LIN {X 0,Y 68.239,Z 470.992,A -85,B 0,C 180,E1 -29740.841,E2 -29740.841} C_VEL
LIN {X 0,Y 69.162,Z 475.21,A -85,B 0,C 180,E1 -29748.344,E2 -29748.344} C_VEL
LIN {X 0,Y 69.85,Z 480.054,A -85,B 0,C 180,E1 -29755.151,E2 -29755.151} C_VEL
LIN {X 0,Y 70.329,Z 485.314,A -85,B 0,C 180,E1 -29761.664,E2 -29761.664} C_VEL
LIN {X 0,Y 70.246,Z 486.749,A -85,B 0,C 180,E1 -29763.244,E2 -29763.244} C_VEL
LIN {X 0,Y 62.959,Z 496.336,A -85,B 0,C 180,E1 -29768.731,E2 -29768.731} C_VEL
LIN {X 0,Y 56.259,Z 504.164,A -85,B 0,C 180,E1 -29775.534,E2 -29775.534} C_VEL
LIN {X 0,Y 50.423,Z 510.748,A -85,B 0,C 180,E1 -29784.262,E2 -29784.262} C_VEL
LIN {X 0,Y 45.973,Z 515.938,A -85,B 0,C 180,E1 -29794.386,E2 -29794.386} C_VEL
LIN {X 0,Y 42.364,Z 521.062,A -85,B 0,C 180,E1 -29809.38,E2 -29809.38} C_VEL
LIN {X 0,Y 41.451,Z 524.116,A -85,B 0,C 180,E1 -29822.031,E2 -29822.031} C_VEL
LIN {X 0,Y 43.45,Z 527.149,A -85,B 0,C 180,E1 -29839.683,E2 -29839.683} C_VEL
LIN {X 0,Y 48.615,Z 528.811,A -85,B 0,C 180,E1 -29854.297,E2 -29854.297} C_VEL
LIN {X 0,Y 55.931,Z 529.259,A -85,B 0,C 180,E1 -29865.444,E2 -29865.444} C_VEL
LIN {X 0,Y 64.604,Z 528.582,A -85,B 0,C 180,E1 -29873.754,E2 -29873.754} C_VEL
LIN {X 0,Y 74.136,Z 526.812,A -85,B 0,C 180,E1 -29879.999,E2 -29879.999} C_VEL
LIN {X 0,Y 84.097,Z 523.976,A -85,B 0,C 180,E1 -29884.595,E2 -29884.595} C_VEL
LIN {X 0,Y 85.983,Z 523.37,A -85,B 0,C 180,E1 -29885.95,E2 -29885.95} C_VEL
LIN {X 0,Y 87.239,Z 522.957,A -85,B 0,C 180,E1 -29888.38,E2 -29888.38} C_VEL
LIN {X 0,Y 87.487,Z 522.949,A -85,B 0,C 180,E1 -29891.862,E2 -29891.862} C_VEL
LIN {X 0,Y 87.094,Z 523.267,A -85,B 0,C 180,E1 -29894.695,E2 -29894.695} C_VEL
LIN {X 0,Y 86.771,Z 523.554,A -85,B 0,C 180,E1 -29896.465,E2 -29896.465} C_VEL
LIN {X 0,Y 84.907,Z 524.361,A -85,B 0,C 180,E1 -29897.846,E2 -29897.846} C_VEL
LIN {X 0,Y 75.254,Z 527.595,A -85,B 0,C 180,E1 -29900.948,E2 -29900.948} C_VEL
LIN {X 0,Y 63.005,Z 530.583,A -85,B 0,C 180,E1 -29906.826,E2 -29906.826} C_VEL
LIN {X 0,Y 51.75,Z 532.139,A -85,B 0,C 180,E1 -29915.426,E2 -29915.426} C_VEL
LIN {X 0,Y 42.308,Z 532.255,A -85,B 0,C 180,E1 -29928.357,E2 -29928.357} C_VEL
LIN {X 0,Y 36.34,Z 531.011,A -85,B 0,C 180,E1 -29947.243,E2 -29947.243} C_VEL
LIN {X 0,Y 35.092,Z 529.839,A -85,B 0,C 180,E1 -29958.444,E2 -29958.444} C_VEL
LIN {X 0,Y 35.123,Z 528.239,A -85,B 0,C 180,E1 -29969.997,E2 -29969.997} C_VEL
LIN {X 0,Y 35.704,Z 524.788,A -85,B 0,C 180,E1 -29987.17,E2 -29987.17} C_VEL
LIN {X 0,Y 38.996,Z 520.194,A -85,B 0,C 180,E1 -30002.726,E2 -30002.726} C_VEL
LIN {X 0,Y 45.724,Z 513.255,A -85,B 0,C 180,E1 -30016.89,E2 -30016.89} C_VEL
LIN {X 0,Y 53.05,Z 505.696,A -85,B 0,C 180,E1 -30025.889,E2 -30025.889} C_VEL
LIN {X 0,Y 56.999,Z 501.154,A -85,B 0,C 180,E1 -30029.662,E2 -30029.662} C_VEL
LIN {X 0,Y 61.398,Z 493.41,A -85,B 0,C 180,E1 -30036.302,E2 -30036.302} C_VEL
LIN {X 0,Y 63.78,Z 488.74,A -85,B 0,C 180,E1 -30039.696,E2 -30039.696} C_VEL
LIN {X 0,Y 64.398,Z 483.456,A -85,B 0,C 180,E1 -30045.786,E2 -30045.786} C_VEL
LIN {X 0,Y 64.825,Z 478.418,A -85,B 0,C 180,E1 -30052.055,E2 -30052.055} C_VEL
LIN {X 0,Y 64.92,Z 477.146,A -85,B 0,C 180,E1 -30053.786,E2 -30053.786} C_VEL
LIN {X 0,Y 64.579,Z 474.051,A -85,B 0,C 180,E1 -30060.001,E2 -30060.001} C_VEL
LIN {X 0,Y 63.893,Z 471.746,A -85,B 0,C 180,E1 -30068.141,E2 -30068.141} C_VEL
LIN {X 0,Y 63.705,Z 471.009,A -85,B 0,C 180,E1 -30072.747,E2 -30072.747} C_VEL
LIN {X 0,Y 63.211,Z 471.361,A -85,B 0,C 180,E1 -30079.485,E2 -30079.485} C_VEL
LIN {X 0,Y 63.047,Z 472.618,A -85,B 0,C 180,E1 -30086.907,E2 -30086.907} C_VEL
LIN {X 0,Y 63.522,Z 474.951,A -85,B 0,C 180,E1 -30095.851,E2 -30095.851} C_VEL
LIN {X 0,Y 63.895,Z 477.2,A -85,B 0,C 180,E1 -30101.298,E2 -30101.298} C_VEL
LIN {X 0,Y 64.259,Z 480.2,A -85,B 0,C 180,E1 -30107.059,E2 -30107.059} C_VEL
LIN {X 0,Y 64.466,Z 484.389,A -85,B 0,C 180,E1 -30113.662,E2 -30113.662} C_VEL
LIN {X 0,Y 64.505,Z 488.05,A -85,B 0,C 180,E1 -30118.836,E2 -30118.836} C_VEL
LIN {X 0,Y 63.381,Z 489.883,A -85,B 0,C 180,E1 -30120.07,E2 -30120.07} C_VEL
LIN {X 0,Y 55.729,Z 498.916,A -85,B 0,C 180,E1 -30125.807,E2 -30125.807} C_VEL
LIN {X 0,Y 48.757,Z 506.356,A -85,B 0,C 180,E1 -30133.247,E2 -30133.247} C_VEL
LIN {X 0,Y 42.447,Z 512.783,A -85,B 0,C 180,E1 -30143.439,E2 -30143.439} C_VEL
LIN {X 0,Y 38.014,Z 517.582,A -85,B 0,C 180,E1 -30155.306,E2 -30155.306} C_VEL
LIN {X 0,Y 34.671,Z 522.492,A -85,B 0,C 180,E1 -30173.919,E2 -30173.919} C_VEL
LIN {X 0,Y 34.527,Z 525.01,A -85,B 0,C 180,E1 -30187.639,E2 -30187.639} C_VEL
LIN {X 0,Y 37.457,Z 527.626,A -85,B 0,C 180,E1 -30205.743,E2 -30205.743} C_VEL
LIN {X 0,Y 44.328,Z 529.337,A -85,B 0,C 180,E1 -30222.045,E2 -30222.045} C_VEL
LIN {X 0,Y 52.33,Z 529.729,A -85,B 0,C 180,E1 -30232.281,E2 -30232.281} C_VEL
LIN {X 0,Y 63.259,Z 528.907,A -85,B 0,C 180,E1 -30240.821,E2 -30240.821} C_VEL
LIN {X 0,Y 72.278,Z 527.298,A -85,B 0,C 180,E1 -30245.579,E2 -30245.579} C_VEL
LIN {X 0,Y 83.302,Z 524.325,A -85,B 0,C 180,E1 -30249.714,E2 -30249.714} C_VEL
LIN {X 0,Y 85.768,Z 523.476,A -85,B 0,C 180,E1 -30250.483,E2 -30250.483} C_VEL
LIN {X 0,Y 87.552,Z 522.917,A -85,B 0,C 180,E1 -30252.094,E2 -30252.094} C_VEL
LIN {X 0,Y 87.094,Z 523.267,A -85,B 0,C 180,E1 -30254.695,E2 -30254.695} C_VEL
LIN {X 0,Y 86.085,Z 523.782,A -85,B 0,C 180,E1 -30256.223,E2 -30256.223} C_VEL
LIN {X 0,Y 83.521,Z 524.843,A -85,B 0,C 180,E1 -30257.731,E2 -30257.731} C_VEL
LIN {X 0,Y 79.236,Z 526.3,A -85,B 0,C 180,E1 -30258.909,E2 -30258.909} C_VEL
LIN {X 0,Y 75.495,Z 527.361,A -85,B 0,C 180,E1 -30259.378,E2 -30259.378} C_VEL
LIN {X 0,Y 64.083,Z 529.81,A -85,B 0,C 180,E1 -30260.093,E2 -30260.093} C_VEL
LIN {X 0,Y 58.606,Z 530.639,A -85,B 0,C 180,E1 -30261.55,E2 -30261.55} C_VEL
LIN {X 0,Y 57.584,Z 530.755,A -85,B 0,C 180,E1 -30262.052,E2 -30262.052} C_VEL
LIN {X 0,Y 47.968,Z 531.742,A -85,B 0,C 180,E1 -30268.465,E2 -30268.465} C_VEL
LIN {X 0,Y 37.285,Z 531.697,A -85,B 0,C 180,E1 -30281.061,E2 -30281.061} C_VEL
LIN {X 0,Y 29.932,Z 530.261,A -85,B 0,C 180,E1 -30301.989,E2 -30301.989} C_VEL
LIN {X 0,Y 28.199,Z 528.973,A -85,B 0,C 180,E1 -30315.565,E2 -30315.565} C_VEL
LIN {X 0,Y 28.043,Z 527.294,A -85,B 0,C 180,E1 -30329.996,E2 -30329.996} C_VEL
LIN {X 0,Y 28.995,Z 523.679,A -85,B 0,C 180,E1 -30351.316,E2 -30351.316} C_VEL
LIN {X 0,Y 33.235,Z 518.91,A -85,B 0,C 180,E1 -30369.37,E2 -30369.37} C_VEL
LIN {X 0,Y 39.922,Z 512.879,A -85,B 0,C 180,E1 -30382.385,E2 -30382.385} C_VEL
LIN {X 0,Y 47.972,Z 505.34,A -85,B 0,C 180,E1 -30391.516,E2 -30391.516} C_VEL
LIN {X 0,Y 50.877,Z 502.415,A -85,B 0,C 180,E1 -30393.874,E2 -30393.874} C_VEL
LIN {X 0,Y 53.428,Z 498.975,A -85,B 0,C 180,E1 -30397.035,E2 -30397.035} C_VEL
LIN {X 0,Y 57.849,Z 491.973,A -85,B 0,C 180,E1 -30402.88,E2 -30402.88} C_VEL
LIN {X 0,Y 58.451,Z 490.648,A -85,B 0,C 180,E1 -30404.124,E2 -30404.124} C_VEL
LIN {X 0,Y 59.603,Z 485.201,A -85,B 0,C 180,E1 -30411.247,E2 -30411.247} C_VEL
LIN {X 0,Y 60.222,Z 481.579,A -85,B 0,C 180,E1 -30416.656,E2 -30416.656} C_VEL
LIN {X 0,Y 60.25,Z 480.054,A -85,B 0,C 180,E1 -30420.001,E2 -30420.001} C_VEL
LIN {X 0,Y 59.924,Z 478.006,A -85,B 0,C 180,E1 -30426.736,E2 -30426.736} C_VEL
LIN {X 0,Y 59.645,Z 477,A -85,B 0,C 180,E1 -30433.631,E2 -30433.631} C_VEL
LIN {X 0,Y 59.095,Z 477.547,A -85,B 0,C 180,E1 -30440.904,E2 -30440.904} C_VEL
LIN {X 0,Y 58.901,Z 478.853,A -85,B 0,C 180,E1 -30448.508,E2 -30448.508} C_VEL
LIN {X 0,Y 59.072,Z 480.036,A -85,B 0,C 180,E1 -30453.616,E2 -30453.616} C_VEL
LIN {X 0,Y 59.17,Z 482.171,A -85,B 0,C 180,E1 -30459.622,E2 -30459.622} C_VEL
LIN {X 0,Y 59.182,Z 485.792,A -85,B 0,C 180,E1 -30467.178,E2 -30467.178} C_VEL
LIN {X 0,Y 58.934,Z 489.465,A -85,B 0,C 180,E1 -30473.401,E2 -30473.401} C_VEL
LIN {X 0,Y 58.419,Z 490.884,A -85,B 0,C 180,E1 -30475.152,E2 -30475.152} C_VEL
LIN {X 0,Y 50.26,Z 499.834,A -85,B 0,C 180,E1 -30480.701,E2 -30480.701} C_VEL
LIN {X 0,Y 42.699,Z 507.2,A -85,B 0,C 180,E1 -30488.267,E2 -30488.267} C_VEL
LIN {X 0,Y 35.769,Z 513.506,A -85,B 0,C 180,E1 -30499.251,E2 -30499.251} C_VEL
LIN {X 0,Y 30.083,Z 519.007,A -85,B 0,C 180,E1 -30515.94,E2 -30515.94} C_VEL
LIN {X 0,Y 27.26,Z 523.794,A -85,B 0,C 180,E1 -30541.043,E2 -30541.043} C_VEL
LIN {X 0,Y 28.364,Z 526.16,A -85,B 0,C 180,E1 -30558.021,E2 -30558.021} C_VEL
LIN {X 0,Y 31.985,Z 528.09,A -85,B 0,C 180,E1 -30573.929,E2 -30573.929} C_VEL
LIN {X 0,Y 39.937,Z 529.739,A -85,B 0,C 180,E1 -30589.863,E2 -30589.863} C_VEL
LIN {X 0,Y 49.591,Z 530.2,A -85,B 0,C 180,E1 -30599.999,E2 -30599.999} C_VEL
LIN {X 0,Y 60.087,Z 529.55,A -85,B 0,C 180,E1 -30606.716,E2 -30606.716} C_VEL
LIN {X 0,Y 71.745,Z 527.672,A -85,B 0,C 180,E1 -30611.596,E2 -30611.596} C_VEL
LIN {X 0,Y 78.218,Z 526.098,A -85,B 0,C 180,E1 -30613.576,E2 -30613.576} C_VEL
LIN {X 0,Y 74.855,Z 527.129,A -85,B 0,C 180,E1 -30615.194,E2 -30615.194} C_VEL
LIN {X 0,Y 61.695,Z 530.146,A -85,B 0,C 180,E1 -30619.983,E2 -30619.983} C_VEL
LIN {X 0,Y 57.584,Z 530.755,A -85,B 0,C 180,E1 -30622.052,E2 -30622.052} C_VEL
LIN {X 0,Y 52.182,Z 531.388,A -85,B 0,C 180,E1 -30624.479,E2 -30624.479} C_VEL
LIN {X 0,Y 42.632,Z 531.649,A -85,B 0,C 180,E1 -30627.711,E2 -30627.711} C_VEL
LIN {X 0,Y 33.336,Z 531.161,A -85,B 0,C 180,E1 -30632.886,E2 -30632.886} C_VEL
LIN {X 0,Y 28.652,Z 530.554,A -85,B 0,C 180,E1 -30639.477,E2 -30639.477} C_VEL
LIN {X 0,Y 23.914,Z 529.462,A -85,B 0,C 180,E1 -30653.997,E2 -30653.997} C_VEL
LIN {X 0,Y 21.433,Z 528.092,A -85,B 0,C 180,E1 -30670.854,E2 -30670.854} C_VEL
LIN {X 0,Y 20.982,Z 526.328,A -85,B 0,C 180,E1 -30689.995,E2 -30689.995} C_VEL
LIN {X 0,Y 22.522,Z 522.526,A -85,B 0,C 180,E1 -30717.904,E2 -30717.904} C_VEL
LIN {X 0,Y 28.109,Z 517.57,A -85,B 0,C 180,E1 -30738.589,E2 -30738.589} C_VEL
LIN {X 0,Y 36.03,Z 511.323,A -85,B 0,C 180,E1 -30751.366,E2 -30751.366} C_VEL
LIN {X 0,Y 45.015,Z 503.462,A -85,B 0,C 180,E1 -30759.505,E2 -30759.505} C_VEL
LIN {X 0,Y 47.584,Z 500.852,A -85,B 0,C 180,E1 -30761.593,E2 -30761.593} C_VEL
LIN {X 0,Y 53.082,Z 493.385,A -85,B 0,C 180,E1 -30768.163,E2 -30768.163} C_VEL
LIN {X 0,Y 54.553,Z 489.076,A -85,B 0,C 180,E1 -30774.456,E2 -30774.456} C_VEL
LIN {X 0,Y 54.989,Z 487.813,A -85,B 0,C 180,E1 -30776.337,E2 -30776.337} C_VEL
LIN {X 0,Y 55.486,Z 485.848,A -85,B 0,C 180,E1 -30780.001,E2 -30780.001} C_VEL
LIN {X 0,Y 55.531,Z 484.136,A -85,B 0,C 180,E1 -30785.213,E2 -30785.213} C_VEL
LIN {X 0,Y 55.539,Z 483.612,A -85,B 0,C 180,E1 -30787.271,E2 -30787.271} C_VEL
LIN {X 0,Y 55.276,Z 482.773,A -85,B 0,C 180,E1 -30794.732,E2 -30794.732} C_VEL
LIN {X 0,Y 54.46,Z 483.962,A -85,B 0,C 180,E1 -30805.406,E2 -30805.406} C_VEL
LIN {X 0,Y 54.413,Z 485.611,A -85,B 0,C 180,E1 -30813.486,E2 -30813.486} C_VEL
LIN {X 0,Y 54.157,Z 488.009,A -85,B 0,C 180,E1 -30820.457,E2 -30820.457} C_VEL
LIN {X 0,Y 53.703,Z 491.02,A -85,B 0,C 180,E1 -30826.992,E2 -30826.992} C_VEL
LIN {X 0,Y 53.519,Z 492.025,A -85,B 0,C 180,E1 -30828.963,E2 -30828.963} C_VEL
LIN {X 0,Y 52.201,Z 493.759,A -85,B 0,C 180,E1 -30830.248,E2 -30830.248} C_VEL
LIN {X 0,Y 43.86,Z 501.992,A -85,B 0,C 180,E1 -30835.407,E2 -30835.407} C_VEL
LIN {X 0,Y 35.513,Z 509.238,A -85,B 0,C 180,E1 -30843.563,E2 -30843.563} C_VEL
LIN {X 0,Y 26.954,Z 516.081,A -85,B 0,C 180,E1 -30858.727,E2 -30858.727} C_VEL
LIN {X 0,Y 21.491,Z 521.012,A -85,B 0,C 180,E1 -30881.162,E2 -30881.162} C_VEL
LIN {X 0,Y 20.551,Z 525.067,A -85,B 0,C 180,E1 -30913.159,E2 -30913.159} C_VEL
LIN {X 0,Y 23.58,Z 527.234,A -85,B 0,C 180,E1 -30933.406,E2 -30933.406} C_VEL
LIN {X 0,Y 28.742,Z 528.874,A -85,B 0,C 180,E1 -30947.992,E2 -30947.992} C_VEL
LIN {X 0,Y 37.085,Z 530.195,A -85,B 0,C 180,E1 -30959.999,E2 -30959.999} C_VEL
LIN {X 0,Y 49.898,Z 530.66,A -85,B 0,C 180,E1 -30969.614,E2 -30969.614} C_VEL
LIN {X 0,Y 57.76,Z 530.167,A -85,B 0,C 180,E1 -30973.24,E2 -30973.24} C_VEL
LIN {X 0,Y 58.721,Z 530.092,A -85,B 0,C 180,E1 -30973.849,E2 -30973.849} C_VEL
LIN {X 0,Y 45.007,Z 531.349,A -85,B 0,C 180,E1 -30980.458,E2 -30980.458} C_VEL
LIN {X 0,Y 33.047,Z 531.105,A -85,B 0,C 180,E1 -30991.712,E2 -30991.712} C_VEL
LIN {X 0,Y 28.652,Z 530.554,A -85,B 0,C 180,E1 -30999.477,E2 -30999.477} C_VEL
LIN {X 0,Y 24.531,Z 529.769,A -85,B 0,C 180,E1 -31008.504,E2 -31008.504} C_VEL
LIN {X 0,Y 20.423,Z 528.566,A -85,B 0,C 180,E1 -31019.116,E2 -31019.116} C_VEL
LIN {X 0,Y 14.603,Z 525.174,A -85,B 0,C 180,E1 -31052.839,E2 -31052.839} C_VEL
LIN {X 0,Y 15.412,Z 522.318,A -85,B 0,C 180,E1 -31081.829,E2 -31081.829} C_VEL
LIN {X 0,Y 21.253,Z 518.011,A -85,B 0,C 180,E1 -31105.752,E2 -31105.752} C_VEL
LIN {X 0,Y 30.058,Z 511.994,A -85,B 0,C 180,E1 -31119.259,E2 -31119.259} C_VEL
LIN {X 0,Y 39.721,Z 504.468,A -85,B 0,C 180,E1 -31126.673,E2 -31126.673} C_VEL
LIN {X 0,Y 43.028,Z 501.52,A -85,B 0,C 180,E1 -31128.508,E2 -31128.508} C_VEL
LIN {X 0,Y 47.08,Z 496.868,A -85,B 0,C 180,E1 -31132.711,E2 -31132.711} C_VEL
LIN {X 0,Y 48.467,Z 495.008,A -85,B 0,C 180,E1 -31134.445,E2 -31134.445} C_VEL
LIN {X 0,Y 50.072,Z 491.699,A -85,B 0,C 180,E1 -31140.001,E2 -31140.001} C_VEL
LIN {X 0,Y 50.675,Z 489.959,A -85,B 0,C 180,E1 -31143.977,E2 -31143.977} C_VEL
LIN {X 0,Y 50.824,Z 488.946,A -85,B 0,C 180,E1 -31147.949,E2 -31147.949} C_VEL
LIN {X 0,Y 50.68,Z 488.316,A -85,B 0,C 180,E1 -31153.911,E2 -31153.911} C_VEL
LIN {X 0,Y 49.75,Z 489.339,A -85,B 0,C 180,E1 -31165.076,E2 -31165.076} C_VEL
LIN {X 0,Y 49.538,Z 490.507,A -85,B 0,C 180,E1 -31171.66,E2 -31171.66} C_VEL
LIN {X 0,Y 48.857,Z 493.056,A -85,B 0,C 180,E1 -31179.782,E2 -31179.782} C_VEL
LIN {X 0,Y 48.308,Z 494.617,A -85,B 0,C 180,E1 -31183.334,E2 -31183.334} C_VEL
LIN {X 0,Y 39.127,Z 503.053,A -85,B 0,C 180,E1 -31187.706,E2 -31187.706} C_VEL
LIN {X 0,Y 28.638,Z 511.224,A -85,B 0,C 180,E1 -31196.49,E2 -31196.49} C_VEL
LIN {X 0,Y 20.591,Z 516.76,A -85,B 0,C 180,E1 -31210.048,E2 -31210.048} C_VEL
LIN {X 0,Y 14.209,Z 521.495,A -85,B 0,C 180,E1 -31238.405,E2 -31238.405} C_VEL
LIN {X 0,Y 15.15,Z 526.03,A -85,B 0,C 180,E1 -31292.358,E2 -31292.358} C_VEL
LIN {X 0,Y 24.297,Z 528.986,A -85,B 0,C 180,E1 -31319.998,E2 -31319.998} C_VEL
LIN {X 0,Y 37.712,Z 530.853,A -85,B 0,C 180,E1 -31332.81,E2 -31332.81} C_VEL
LIN {X 0,Y 36.393,Z 530.86,A -85,B 0,C 180,E1 -31335.075,E2 -31335.075} C_VEL
LIN {X 0,Y 23.905,Z 529.721,A -85,B 0,C 180,E1 -31348.109,E2 -31348.109} C_VEL
LIN {X 0,Y 14.95,Z 527.199,A -85,B 0,C 180,E1 -31381.952,E2 -31381.952} C_VEL
LIN {X 0,Y 13.916,Z 525.31,A -85,B 0,C 180,E1 -31409.993,E2 -31409.993} C_VEL
LIN {X 0,Y 15.412,Z 522.318,A -85,B 0,C 180,E1 -31441.829,E2 -31441.829} C_VEL
LIN {X 0,Y 17.843,Z 519.939,A -85,B 0,C 180,E1 -31458.567,E2 -31458.567} C_VEL
LIN {X 0,Y 22.738,Z 515.343,A -85,B 0,C 180,E1 -31479.524,E2 -31479.524} C_VEL
LIN {X 0,Y 29.115,Z 510.081,A -85,B 0,C 180,E1 -31491.945,E2 -31491.945} C_VEL
LIN {X 0,Y 33.572,Z 506.599,A -85,B 0,C 180,E1 -31495.272,E2 -31495.272} C_VEL
LIN {X 0,Y 40.438,Z 500.992,A -85,B 0,C 180,E1 -31497.793,E2 -31497.793} C_VEL
LIN {X 0,Y 43.001,Z 498.322,A -85,B 0,C 180,E1 -31500.001,E2 -31500.001} C_VEL
LIN {X 0,Y 44.424,Z 496.579,A -85,B 0,C 180,E1 -31502.268,E2 -31502.268} C_VEL
LIN {X 0,Y 45.2,Z 495.379,A -85,B 0,C 180,E1 -31504.46,E2 -31504.46} C_VEL
LIN {X 0,Y 45.807,Z 494.036,A -85,B 0,C 180,E1 -31508.826,E2 -31508.826} C_VEL
LIN {X 0,Y 45.244,Z 493.87,A -85,B 0,C 180,E1 -31518.101,E2 -31518.101} C_VEL
LIN {X 0,Y 44.521,Z 495.027,A -85,B 0,C 180,E1 -31528.268,E2 -31528.268} C_VEL
LIN {X 0,Y 44.247,Z 495.66,A -85,B 0,C 180,E1 -31531.393,E2 -31531.393} C_VEL
LIN {X 0,Y 43.313,Z 497.202,A -85,B 0,C 180,E1 -31535.783,E2 -31535.783} C_VEL
LIN {X 0,Y 33.661,Z 505.338,A -85,B 0,C 180,E1 -31538.784,E2 -31538.784} C_VEL
LIN {X 0,Y 24.337,Z 511.884,A -85,B 0,C 180,E1 -31543.792,E2 -31543.792} C_VEL
LIN {X 0,Y 13.243,Z 518.381,A -85,B 0,C 180,E1 -31557.957,E2 -31557.957} C_VEL
LIN {X 0,Y 5.996,Z 523.517,A -85,B 0,C 180,E1 -31625.899,E2 -31625.899} C_VEL
LIN {X 0,Y 14.171,Z 527.348,A -85,B 0,C 180,E1 -31687.256,E2 -31687.256} C_VEL
LIN {X 0,Y 17.023,Z 528.102,A -85,B 0,C 180,E1 -31691.755,E2 -31691.755} C_VEL
LIN {X 0,Y 14.97,Z 527.781,A -85,B 0,C 180,E1 -31700.106,E2 -31700.106} C_VEL
LIN {X 0,Y 9.335,Z 526.207,A -85,B 0,C 180,E1 -31721.149,E2 -31721.149} C_VEL
LIN {X 0,Y 6.849,Z 524.212,A -85,B 0,C 180,E1 -31769.985,E2 -31769.985} C_VEL
LIN {X 0,Y 11.997,Z 520.042,A -85,B 0,C 180,E1 -31831.469,E2 -31831.469} C_VEL
LIN {X 0,Y 23.218,Z 513.675,A -85,B 0,C 180,E1 -31849.624,E2 -31849.624} C_VEL
LIN {X 0,Y 33.572,Z 506.599,A -85,B 0,C 180,E1 -31855.272,E2 -31855.272} C_VEL
LIN {X 0,Y 35.364,Z 504.986,A -85,B 0,C 180,E1 -31857.147,E2 -31857.147} C_VEL
LIN {X 0,Y 36.878,Z 503.159,A -85,B 0,C 180,E1 -31861.127,E2 -31861.127} C_VEL
LIN {X 0,Y 37.876,Z 501.617,A -85,B 0,C 180,E1 -31865.931,E2 -31865.931} C_VEL
LIN {X 0,Y 38.672,Z 500.285,A -85,B 0,C 180,E1 -31872.447,E2 -31872.447} C_VEL
LIN {X 0,Y 39.267,Z 499.486,A -85,B 0,C 180,E1 -31880.413,E2 -31880.413} C_VEL
LIN {X 0,Y 39.262,Z 499.638,A -85,B 0,C 180,E1 -31886.094,E2 -31886.094} C_VEL
LIN {X 0,Y 39.245,Z 499.674,A -85,B 0,C 180,E1 -31886.447,E2 -31886.447} C_VEL
LIN {X 0,Y 27.551,Z 508.705,A -85,B 0,C 180,E1 -31886.765,E2 -31886.765} C_VEL
LIN {X 0,Y 15.714,Z 515.954,A -85,B 0,C 180,E1 -31886.571,E2 -31886.571} C_VEL
LIN {X 0,Y 5.664,Z 520.85,A -85,B 0,C 180,E1 -31880.494,E2 -31880.494} C_VEL
LIN {X 0,Y 7.089,Z 520.318,A -85,B 0,C 180,E1 -31867.658,E2 -31867.658} C_VEL
LIN {X 0,Y 17.71,Z 515.134,A -85,B 0,C 180,E1 -31867.275,E2 -31867.275} C_VEL
LIN {X 0,Y 28.329,Z 508.635,A -85,B 0,C 180,E1 -31867.136,E2 -31867.136} C_VEL
LIN {X 0,Y 37.9,Z 501.38,A -85,B 0,C 180,E1 -31867.564,E2 -31867.564} C_VEL
LIN {X 0,Y 39.051,Z 500.359,A -85,B 0,C 180,E1 -31868.2,E2 -31868.2} C_VEL
LIN {X 0,Y 40.395,Z 498.974,A -85,B 0,C 180,E1 -31870.021,E2 -31870.021} C_VEL
LIN {X 0,Y 39.712,Z 499.086,A -85,B 0,C 180,E1 -31880.73,E2 -31880.73} C_VEL
LIN {X 0,Y 39.262,Z 499.638,A -85,B 0,C 180,E1 -31886.094,E2 -31886.094} C_VEL
LIN {X 0,Y 39.172,Z 501.616,A -85,B 0,C 180,E1 -31888.585,E2 -31888.585} C_VEL
LIN {X 0,Y 39.172,Z 600,A -85,B 0,C 180,E1 -31888.585,E2 -31888.585} C_VEL
LIN {X 0,Y 39.172,Z 600,A -85,B 0,C 180,E1 -31888.585,E2 -31888.585}

QRS_NEXT_CUT()

QRS_NEXT()
QRS_HOME()

END
